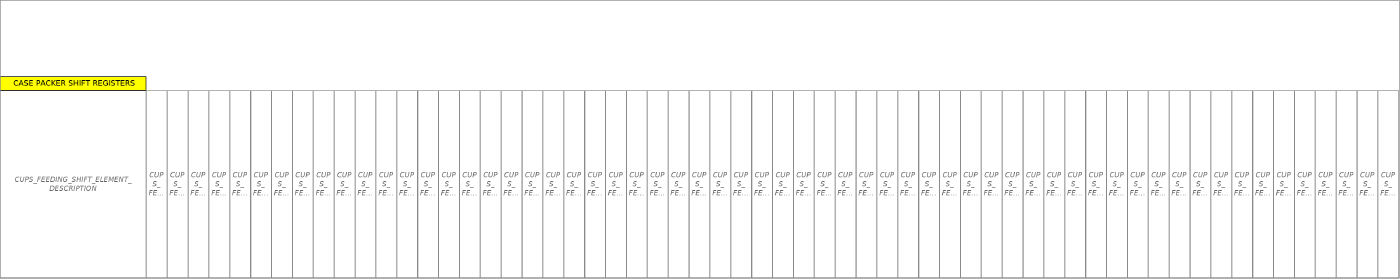
VISUALIZATION CUPS_SHIFT  // 2012x402
    Frame (0,130 210x270)
        shows CUPS_FEEDING_SHIFT_ELEMENT_DESCRIPTION()
    Rectangle (0,110 210x20), "CASE PACKER SHIFT REGISTERS"
    Frame (390,130 30x270)
        shows CUPS_FEEDING_SHIFT_ELEMENT(index := 7)
        shows CUPS_FEEDING_SHIFT_ELEMENT()
    Frame (420,130 30x270)
        shows CUPS_FEEDING_SHIFT_ELEMENT(index := 8)
    Frame (450,130 30x270)
        shows CUPS_FEEDING_SHIFT_ELEMENT(index := 9)
    Frame (480,130 30x270)
        shows CUPS_FEEDING_SHIFT_ELEMENT(index := 10)
    Frame (510,130 30x270)
        shows CUPS_FEEDING_SHIFT_ELEMENT(index := 11)
    Frame (540,130 30x270)
        shows CUPS_FEEDING_SHIFT_ELEMENT(index := 12)
    Frame (570,130 30x270)
        shows CUPS_FEEDING_SHIFT_ELEMENT(index := 13)
    Frame (600,130 30x270)
        shows CUPS_FEEDING_SHIFT_ELEMENT(index := 14)
    Frame (630,130 30x270)
        shows CUPS_FEEDING_SHIFT_ELEMENT(index := 15)
    Frame (660,130 30x270)
        shows CUPS_FEEDING_SHIFT_ELEMENT(index := 16)
    Frame (690,130 30x270)
        shows CUPS_FEEDING_SHIFT_ELEMENT(index := 17)
    Frame (720,130 30x270)
        shows CUPS_FEEDING_SHIFT_ELEMENT(index := 18)
    Frame (750,130 30x270)
        shows CUPS_FEEDING_SHIFT_ELEMENT(index := 19)
    Frame (780,130 30x270)
        shows CUPS_FEEDING_SHIFT_ELEMENT(index := 20)
    Frame (810,130 30x270)
        shows CUPS_FEEDING_SHIFT_ELEMENT(index := 21)
    Frame (840,130 30x270)
        shows CUPS_FEEDING_SHIFT_ELEMENT(index := 22)
    Frame (870,130 30x270)
        shows CUPS_FEEDING_SHIFT_ELEMENT(index := 23)
    Frame (900,130 30x270)
        shows CUPS_FEEDING_SHIFT_ELEMENT(index := 24)
    Frame (930,130 30x270)
        shows CUPS_FEEDING_SHIFT_ELEMENT(index := 25)
    Frame (960,130 30x270)
        shows CUPS_FEEDING_SHIFT_ELEMENT(index := 26)
    Frame (990,130 30x270)
        shows CUPS_FEEDING_SHIFT_ELEMENT(index := 27)
    Frame (1020,130 30x270)
        shows CUPS_FEEDING_SHIFT_ELEMENT(index := 28)
    Frame (1050,130 30x270)
        shows CUPS_FEEDING_SHIFT_ELEMENT(index := 29)
    Frame (1080,130 30x270)
        shows CUPS_FEEDING_SHIFT_ELEMENT(index := 30)
    Frame (1110,130 30x270)
        shows CUPS_FEEDING_SHIFT_ELEMENT(index := 31)
    Frame (1140,130 30x270)
        shows CUPS_FEEDING_SHIFT_ELEMENT(index := 32)
    Frame (1170,130 30x270)
        shows CUPS_FEEDING_SHIFT_ELEMENT(index := 33)
    Frame (1200,130 30x270)
        shows CUPS_FEEDING_SHIFT_ELEMENT(index := 34)
    Frame (1230,130 30x270)
        shows CUPS_FEEDING_SHIFT_ELEMENT(index := 35)
    Frame (1260,130 30x270)
        shows CUPS_FEEDING_SHIFT_ELEMENT(index := 36)
    Frame (1290,130 30x270)
        shows CUPS_FEEDING_SHIFT_ELEMENT(index := 37)
    Frame (1320,130 30x270)
        shows CUPS_FEEDING_SHIFT_ELEMENT(index := 38)
    Frame (1350,130 30x270)
        shows CUPS_FEEDING_SHIFT_ELEMENT(index := 39)
    Frame (1380,130 30x270)
        shows CUPS_FEEDING_SHIFT_ELEMENT(index := 40)
    Frame (1410,130 30x270)
        shows CUPS_FEEDING_SHIFT_ELEMENT(index := 41)
    Frame (1440,130 30x270)
        shows CUPS_FEEDING_SHIFT_ELEMENT(index := 42)
    Frame (1470,130 30x270)
        shows CUPS_FEEDING_SHIFT_ELEMENT(index := 43)
    Frame (1500,130 30x270)
        shows CUPS_FEEDING_SHIFT_ELEMENT(index := 44)
    Frame (1530,130 30x270)
        shows CUPS_FEEDING_SHIFT_ELEMENT(index := 45)
    Frame (1560,130 30x270)
        shows CUPS_FEEDING_SHIFT_ELEMENT(index := 46)
    Frame (1590,130 30x270)
        shows CUPS_FEEDING_SHIFT_ELEMENT(index := 47)
    Frame (1620,130 30x270)
        shows CUPS_FEEDING_SHIFT_ELEMENT(index := 48)
    Frame (1650,130 30x270)
        shows CUPS_FEEDING_SHIFT_ELEMENT(index := 49)
    Frame (1680,130 30x270)
        shows CUPS_FEEDING_SHIFT_ELEMENT(index := 50)
    Frame (1710,130 30x270)
        shows CUPS_FEEDING_SHIFT_ELEMENT(index := 51)
    Frame (1740,130 30x270)
        shows CUPS_FEEDING_SHIFT_ELEMENT(index := 52)
    Frame (1770,130 30x270)
        shows CUPS_FEEDING_SHIFT_ELEMENT(index := 53)
    Frame (1800,130 30x270)
        shows CUPS_FEEDING_SHIFT_ELEMENT(index := 54)
    Frame (1830,130 30x270)
        shows CUPS_FEEDING_SHIFT_ELEMENT(index := 55)
    Frame (1860,130 30x270)
        shows CUPS_FEEDING_SHIFT_ELEMENT(index := 56)
    Frame (1890,130 30x270)
        shows CUPS_FEEDING_SHIFT_ELEMENT(index := 57)
    Frame (1920,130 30x270)
        shows CUPS_FEEDING_SHIFT_ELEMENT(index := 58)
    Frame (1950,130 30x270)
        shows CUPS_FEEDING_SHIFT_ELEMENT(index := 59)
    Frame (1980,130 30x270)
        shows CUPS_FEEDING_SHIFT_ELEMENT(index := 60)
    Frame (210,130 30x270)
        shows CUPS_FEEDING_SHIFT_ELEMENT(index := 1)
        shows CUPS_FEEDING_SHIFT_ELEMENT()
    Frame (240,130 30x270)
        shows CUPS_FEEDING_SHIFT_ELEMENT(index := 2)
        shows CUPS_FEEDING_SHIFT_ELEMENT()
    Frame (270,130 30x270)
        shows CUPS_FEEDING_SHIFT_ELEMENT(index := 3)
        shows CUPS_FEEDING_SHIFT_ELEMENT()
    Frame (300,130 30x270)
        shows CUPS_FEEDING_SHIFT_ELEMENT(index := 4)
        shows CUPS_FEEDING_SHIFT_ELEMENT()
    Frame (330,130 30x270)
        shows CUPS_FEEDING_SHIFT_ELEMENT(index := 5)
        shows CUPS_FEEDING_SHIFT_ELEMENT()
    Frame (360,130 30x270)
        shows CUPS_FEEDING_SHIFT_ELEMENT(index := 6)
        shows CUPS_FEEDING_SHIFT_ELEMENT()
END_VISUALIZATION

(* stored: Version 1.1.0.1, ProductVersion 3.1.4024.3
   Visu CUPS_SHIFT: Id {c4f2a628-3005-4e52-a8d6-5ca42c12fd18} *)
